FUNCTION_BLOCK FB_GantryXYZ EXTENDS FB_PackML_BaseModule 
VAR
    // Sub module definitions here

    // List of sub modules
    ipSubModules_Init : ARRAY[1..Parameters_PackML_Base.MAX_NO_OF_SUBMODULES] OF I_PackML_BaseModule := [];

    // Component definitions here
    AxisX       		: FB_Component_BasicAxis 		:= (Name := 'AxisX');
    AxisY    			: FB_Component_BasicAxis 		:= (Name := 'AxisY');
	AxisZ				: FB_Component_BasicAxis		:= (Name := 'AxisZ');
    GantryCylinder		: FB_GantryXYCylinder			:= (Name := 'Cylinder');

    //Alarms for this module
    GantryAlarms : ARRAY[1..GANTRY_ALARM_COUNT] OF FB_TcAlarm;

	//IO
	LimitSwitchX :BOOL;
	LimitSwitchY :BOOL;
	LimitSwitchZ :BOOL;

	HomeComplete :BOOL;
	


END_VAR

VAR CONSTANT
    GANTRY_ALARM_COUNT : INT := 5;
END_VAR

METHOD PROTECTED Clearing
VAR
	i				: UDINT;
	SubModulesReady : BOOL := TRUE;
END_VAR
CASE SequenceState OF
    0:
        NoStateTasksToComplete := FALSE;
        SequenceState          := SequenceState + 10;
    10:
        //Reset any alarms that get latched
        GantryAlarms[E_Gantry.StartTimeout].Clear(0, 0);
        SequenceState := SequenceState + 10;
    20:
        // Enable here
        AxisX.Enable();
        AxisY.Enable();
		AxisZ.Enable();

        // Check enabled here
        IF AxisX.Enabled AND AxisY.Enabled AND AxisZ.Enabled THEN
            SequenceState := SequenceState + 10;
        END_IF
    30:
        StateTasksComplete := TRUE;
END_CASE

SUPER^.Clearing();
END_METHOD

METHOD PROTECTED CreateEvents
VAR_INPUT
END_VAR
// Add your event creation here
F_CreateAllEventsInClass(Alarms     := GantryAlarms,
                         ClassSize  := SIZEOF(TC_EVENTS.Gantry),
                         pInitEvent := ADR(TC_EVENTS.Gantry.InitReferenceEvent),
                         Prefix     := _Name);

// Super call to base
SUPER^.CreateEvents();
END_METHOD

METHOD CuttingBoxFiveSides : BOOL

VAR_INST
	Step : INT ;	
END_VAR

(*
	F			H
	|			|
D---+-----------+---C
	|			|
	|			| 
B---+-----------+---A
	|			|
	E			G
*)
	CASE Step OF
		
		0:  //Print Info
			
			Trace('Start Cutting Box Five Sides');
			
			Step := Step + 10;	

		10:	//Set Speed
			
			AxisX.Velocity := 10; 
			AxisY.Velocity := 10;
			AxisZ.Velocity := 5;
			
			Step := Step + 10;

		20:	//Positioning Motion to A
   			
			AxisX.MoveAbsolute(0,0);
			AxisY.MoveAbsolute(250,0);		
			
			Step := Step + 10; 
		
		30: //Set Cutting Height
			
			AxisZ.MoveAbsolute(-30,0);
			
			Step := Step + 10;

		40: //Cutting Motion from A to B
			
			AxisX.MoveAbsolute(500,0);		
			
			Step := Step + 10;
		
		50: //Return from Cutting Height 
			
			AxisZ.MoveAbsolute(50,0);

			Step := Step + 10;
		
		60: //Positioning Motion from B to C
			
			AxisX.MoveAbsolute(0,0);
			AxisY.MoveAbsolute(50,0);
	
			Step := Step + 10;

		70: //Set Cutting Height
		
			AxisZ.MoveAbsolute(0,0);

			Step := Step + 10;

		80: //Cutting Motion from C to D
			
			AxisX.MoveAbsolute(500,0);
			AxisY.MoveAbsolute(50,0);

			Step := Step + 10;

		90: //Return from Cutting Height 
			
			AxisZ.MoveAbsolute(50,0);
			
			Step := Step + 10;

		100: //Positioning Motion from D to E
			
			AxisX.MoveAbsolute(450,0);
			AxisY.MoveAbsolute(300,0);

			Step := Step + 10;
		
		110: //Set Cutting Height 	
			
			AxisZ.MoveAbsolute(0,0);
	
			Step := Step + 10;

		120: //Cutting Motion from E to F

			AxisX.MoveAbsolute(450,0);
			AxisY.MoveAbsolute(0,0);
			
			Step := Step + 10;

		130: //Return from Cutting Height 

			AxisZ.MoveAbsolute(50,0);
			
			Step := Step + 10;

		140: //Positioning Motion from F to G

			AxisX.MoveAbsolute(50,0);
			AxisY.MoveAbsolute(300,0);

			Step := Step + 10;

		150: //Cutting Motion from G to H

			AxisX.MoveAbsolute(50,0);
			AxisY.MoveAbsolute(0,0);

			Step := Step + 10;

		160: //Return from Cutting Height 
	
			AxisZ.MoveAbsolute(50,0);

			Step := Step + 10;

		170: //Return to ZERO

			AxisX.MoveAbsolute(0,0);
			AxisY.MoveAbsolute(0,0);

			
			Trace('Box Five Sides is Cut');
			CuttingBoxFiveSides := TRUE;
			Step := 0;
			
	END_CASE
END_METHOD

METHOD CyclicLogic
VAR_INPUT
END_VAR
IF NOT _InitComplete THEN
    _InitComplete := Initialize();
    RETURN;
END_IF

SUPER^.CyclicLogic();

//Set the current alarm severity for this module
_CurrentAlarmSeverity := F_GetMaxSeverityRaised(Alarms := GantryAlarms, CurrentSeverity := _CurrentAlarmSeverity);

//Simulate Alarm Messaging
END_METHOD

METHOD PROTECTED Execute
CASE _CurrentMode OF

	//=================================PRODUCTION MODE==================================
	E_PMLUnitMode.ePMLUnitMode_Production:
		CASE SequenceState OF
			0:
				NoStateTasksToComplete := TRUE;
				
				IF CuttingBoxFiveSides() THEN
					SequenceState := SequenceState + 10;	
				ELSE
					CuttingBoxFiveSides();
				END_IF		
				
			10:		
				StateTasksComplete := TRUE;
				StateComplete();
			END_CASE

	//=================================MAINTENANCE & MANUAL MODE==================================
	E_PMLUnitMode.ePMLUnitMode_Maintenance, E_PMLUnitMode.ePMLUnitMode_Manual:
		;
END_CASE
END_METHOD

METHOD PROTECTED HMIPermissions
//General Mode Based Monitoring and handling of HMI control
CASE _CurrentMode OF
   
 E_PMLUnitMode.ePMLUnitMode_Production:
        CASE _CurrentState OF
            E_PMLState.ePMLState_Stopped:
				AllowHMIControl(ThisModuleOnly := FALSE);
            E_PMLState.ePMLState_Idle:
				AllowHMIControl(ThisModuleOnly := FALSE);
            E_PMLState.ePMLState_Suspended:
         		AllowHMIControl(ThisModuleOnly := FALSE);
            E_PMLState.ePMLState_Execute:
            	AllowHMIControl(ThisModuleOnly := FALSE); 
            E_PMLState.ePMLState_Aborted:
                AllowHMIControl(ThisModuleOnly := FALSE); 
            E_PMLState.ePMLState_Held:
                AllowHMIControl(ThisModuleOnly := FALSE); 
            E_PMLState.ePMLState_Complete:
          		AllowHMIControl(ThisModuleOnly := FALSE); 
        END_CASE
		
    E_PMLUnitMode.ePMLUnitMode_Manual:
        AllowHMIControl(ThisModuleOnly := FALSE); 
	E_PMLUnitMode.ePMLUnitMode_Maintenance:
        AllowHMIControl(ThisModuleOnly := FALSE); 
END_CASE
END_METHOD

METHOD Homing : BOOL

VAR_INST
	Step : INT ;	
END_VAR
	CASE Step OF
		
		0: 
			Trace(' first line');
			Step := Step + 10; 
		10:
			Trace('HomeY');
			Step := Step + 10;
	
		20:	
			Trace('HomeZ');
			Homing := TRUE;
			Step := 0;	

	END_CASE
END_METHOD

//! @summary Basic module initialization logic
METHOD PROTECTED Initialize : BOOL;
VAR
    i                        : UDINT;
    varInfo                  : __SYSTEM.VAR_INFO;
    AllSubUnitsInitialized   : BOOL := TRUE;
    AllComponentsInitialized : BOOL := TRUE;
END_VAR

//! @description This method is called by <c>CyclicLogic()</c> as required
Initialize := FALSE;
CASE DescendantSequenceState OF
    0:
		RegisterComponent(AxisX);
		RegisterComponent(AxisY);	
		RegisterComponent(AxisZ);	
		RegisterComponent(GantryCylinder);
		
        _LogModeChanges         := FALSE;
        _LogStateChanges        := FALSE;
        DescendantSequenceState := DescendantSequenceState + 10;
    10:
        DescendantSequenceState := DescendantSequenceState + 10;
    20:
        //Copy Mode names
        FOR i := 1 TO 3 DO
            ModeNames[i] := F_UnitModeToString(UDINT_TO_DINT(i));
        END_FOR

        DescendantSequenceState := DescendantSequenceState + 10;
    30:
        //Call the Super
        IF SUPER^.Initialize() THEN
            DescendantSequenceState := DescendantSequenceState + 10;
        END_IF
    40:
        Initialize := TRUE;
END_CASE
END_METHOD

METHOD PROTECTED Resetting
VAR
	i				: UDINT;
	SubModulesReady : BOOL := TRUE;
END_VAR
CASE _CurrentMode OF

	//=================================PRODUCTION MODE==================================
	E_PMLUnitMode.ePMLUnitMode_Production:
		CASE SequenceState OF
			0:
				NoStateTasksToComplete := TRUE;
				
				IF Homing() THEN
					SequenceState := SequenceState + 10;	
				ELSE
					Homing();
				END_IF		
				
			10:		
				StateTasksComplete := TRUE;
				SUPER^.Resetting();
		END_CASE

	//=================================MAINTENANCE & MANUAL MODE==================================
	E_PMLUnitMode.ePMLUnitMode_Maintenance, E_PMLUnitMode.ePMLUnitMode_Manual:
		;
END_CASE
END_METHOD

END_FUNCTION_BLOCK

(* stored: Version 1.1.0.1
   POU FB_GantryXYZ: Id {496b17f1-4b0a-4954-89f4-eec9ef72b2f5}, SpecialFunc None
   Folder MyMethods: Id {df43c4fc-4941-0a05-2048-b885d685c5f2}
   Folder States: Id {83d122fa-7c6a-0e7c-1bbf-3cae8b533243}
   Method Clearing: Id {95c08e6a-01f8-0092-17a5-ee449a2d4d0d}
   Method CreateEvents: Id {4ec0ace2-c308-44b2-84a1-60ba649bd547}
   Method CuttingBoxFiveSides: Id {373688d2-86ff-084a-2e79-b1d27d5776ec}
   Method CyclicLogic: Id {02def406-fced-425b-89cd-43b7d8052b02}
   Method Execute: Id {87781098-e2be-0050-2467-1f830db3673b}
   Method HMIPermissions: Id {a98019a5-2d4d-097b-1c9d-7422486c9b5b}
   Method Homing: Id {72d228ce-b399-0094-138d-59f534ec17d5}
   Method Initialize: Id {b4a0fd62-4385-4420-ae43-9bea35a3f798}
   Method Resetting: Id {e9851c76-6213-0482-2237-5496172b7e77} *)
